TYPE U_MoverFeedback :
UNION
	sName	:ST_MoverFeedback;
	aArray	:ARRAY[0..GVL.MAX_FEEDBACK] OF MC_PlanarFeedback;
END_UNION
END_TYPE
//構造体で記載したFeedbackをUpdateする時にFORで処理できるように、同じ要素数の配列と同期する。

(* stored: Version 1.1.0.1
   DUT U_MoverFeedback: Id {250d10e1-89e0-4534-9568-b21230bb0c46} *)
